Universal Robots PolyScope program: last_test_1.8.urp

ProgramRoot setBeforeStartSequence=true; directory=/programs/KINGSTON; kinematics=(a=[0, -0.425, -0.39225, 0, 0, 0], d=[0.08916, 0, 0, 0.10915, 0.09465, 0.0823], alpha=[1.5708, 0, 0, 1.5708, -1.5708, 0], deltaTheta=[0, 0, 0, 0, 0, 0], status=notInitialized); name=last_test; programVersion=(project__name=PolyScope, major__version=1, minor__version=8, svn__revision=11657, build__date=Oct 09 2013, 20:14:19); robotEnvironmentFileName=default; serialNumberRobot=2013210504
  BeforeStart description=COMMAND_SEQUENCE_BEFORE_PROGRAM_START; name=BeforeStart
    Assignment assignmentValueSource=0; expr=0; operatorValueType=INTEGER; valueSource=EXPRESSION; variable=(name=var_1, prefersPersistentValue=false, requestANewUniqueName=false)
    Assignment assignmentValueSource=0; expr=1; operatorValueType=INTEGER; valueSource=EXPRESSION; variable=(name=var_safety, prefersPersistentValue=false, requestANewUniqueName=false)
    Assignment assignmentValueSource=0; expr=50; operatorValueType=INTEGER; valueSource=EXPRESSION; variable=(name=var_force, prefersPersistentValue=false, requestANewUniqueName=false)
    Assignment assignmentValueSource=0; expr=[1,0]; operatorValueType=INTEGER; valueSource=EXPRESSION; variable=(name=var_moveType, prefersPersistentValue=false, requestANewUniqueName=false)
    Assignment assignmentValueSource=0; expr=[6,0,0,0,0,0,0]; operatorValueType=INTEGER; valueSource=EXPRESSION; variable=(name=receive_data, prefersPersistentValue=false, requestANewUniqueName=false)
    Assignment assignmentValueSource=0; expr=p[0,0,0,0,0,0]; operatorValueType=INTEGER; valueSource=EXPRESSION; variable=(name=Move_To_Pos, prefersPersistentValue=false, requestANewUniqueName=false)
    CallSubProgram subProgramNodeToCall=pose_1=get_forward_kin()
    Suppressed suppressedNode=[5,110,0,40,0,40]
    Comment 
    Suppressed suppressedNode=receive_data=socket_read_ascii_float(5)
    Assignment assignmentValueSource=0; expr=[0.2,0.2]; operatorValueType=INTEGER; valueSource=EXPRESSION; variable=(name=var_velacc, prefersPersistentValue=false, requestANewUniqueName=false)
    Script type=0; expressionBranchNode=socket_open("192.168.10.2",30000)
    Assignment assignmentValueSource=0; expr=[0,0]; operatorValueType=INTEGER; valueSource=EXPRESSION; variable=(name=task, prefersPersistentValue=false, requestANewUniqueName=false)
    Assignment assignmentValueSource=0; expr=0; operatorValueType=INTEGER; valueSource=EXPRESSION; variable=(name=coop, prefersPersistentValue=false, requestANewUniqueName=false)
  MainProgram cartesianAcceleration=1.2; cartesianSpeed=0.25; jointAcceleration=1.3962634015954636; jointSpeed=1.0471975511965976; moveAsFastAsPossible=true; sharedProcessMoveBlendRadius=0.025; featureReference=(installationNameReference=Base); motionType=JOINT_SPACE
    Suppressed suppressedNode=___tran51ate_this_name___Joint_0_name
    Suppressed suppressedNode=1
    Suppressed 
    Suppressed suppressedNode=0
    Script type=0; expressionBranchNode=ExpressionVariableNode=socket_read_ascii_float(1)
    If expr=ExpressionVariableNode[1]≟2; type=IF_NODE
      CallSubProgram subProgramNodeToCall=pose_1=get_forward_kin()
      Assignment assignmentValueSource=0; expr=[0,0]; operatorValueType=INTEGER; valueSource=EXPRESSION; variable=(name=task, prefersPersistentValue=false, requestANewUniqueName=false)
    If expr=task[1]≟3; type=ELSEIF_NODE
      Assignment assignmentValueSource=0; expr=1; operatorValueType=INTEGER; valueSource=EXPRESSION; variable=(name=coop, prefersPersistentValue=false, requestANewUniqueName=false)
      Script type=0; expressionBranchNode=socket_send_string("1")
      Assignment assignmentValueSource=0; expr=[0,0]; operatorValueType=INTEGER; valueSource=EXPRESSION; variable=(name=task, prefersPersistentValue=false, requestANewUniqueName=false)
    If expr=task[1]≟4; type=ELSEIF_NODE
      Assignment assignmentValueSource=0; expr=0; operatorValueType=INTEGER; valueSource=EXPRESSION; variable=(name=coop, prefersPersistentValue=false, requestANewUniqueName=false)
      Script type=0; expressionBranchNode=socket_send_string("1")
      Assignment assignmentValueSource=0; expr=[0,0]; operatorValueType=INTEGER; valueSource=EXPRESSION; variable=(name=task, prefersPersistentValue=false, requestANewUniqueName=false)
    If expr=task[1]≟5; type=ELSEIF_NODE
      CallSubProgram subProgramNodeToCall=receive_data=socket_read_ascii_float(2)
    If expr=task[1]≟6; type=ELSEIF_NODE
      CallSubProgram subProgramNodeToCall=receive_data=socket_read_ascii_float(2)
    If expr=task[1]≟7; type=ELSEIF_NODE
      CallSubProgram subProgramNodeToCall=receive_data=socket_read_ascii_float(2)
    If expr=task[1]≟8; type=ELSEIF_NODE
      CallSubProgram subProgramNodeToCall=receive_data=socket_read_ascii_float(5)
    If expr=task[1]≟1; type=ELSEIF_NODE
      CallSubProgram subProgramNodeToCall=receive_data=socket_read_ascii_float(6)
    Wait analogComparison=0; analogInputRange=0; analogValue=0.0; digitalValue=0; selectedAnalogSensor=-1; selectedDigitalSensor=-1; waitTime=0.01; type=TIMER_WAIT
  SubProgram name=Safety_Program
    Assignment assignmentValueSource=0; expr=0; operatorValueType=INTEGER; valueSource=EXPRESSION; variable=(name=var_safety, prefersPersistentValue=false, requestANewUniqueName=false)
    Move cartesianAcceleration=1.2; cartesianSpeed=0.25; jointAcceleration=1.3962634015954636; jointSpeed=1.0471975511965976; moveAsFastAsPossible=true; sharedProcessMoveBlendRadius=0.025; featureReference=(installationNameReference=Base); motionType=JOINT_SPACE
      Waypoint blendRadius=0.05; cartesianAcceleration=1.2; cartesianSpeed=0.25; jointAcceleration=1.3962634015954636; jointSpeed=0.10471975511965977; nextMotionTime=2.0; stoppoint=true; useSharedBlendParameter=true; position=TCP in base x=-199.996 y=-200 z=249.995 mm, rx=3.1416 ry=0 rz=0 rad; joints [-112.3, -59.43, -107.723, -102.846, 90, -202.3] deg; positionType=RELATIVE_POSITION; waypointPoseInFeatureCoordinates=(pos=(x=-0.19999561252286474, y=-0.2000002740460248, z=0.24999526084687385), rot=(x=3.1415926535838667, y=-2.8424371718740507E-6, z=-5.400202873880619E-6)); name=Waypoint_1; relativeFromJointPositionVector=(joint=[-1.96001, -1.01639, -2.01843, -1.67755, 1.5708, -3.53081], isUndefined=false); relativeFromToolAxisAngle=(x=-3.141579017620853, y=5.64237603120038E-5, z=-8.76472952232187E-6); relativeFromToolPosition=(x=-0.20000006548800986, y=-0.19998241022118884, z=0.19999450290156112)
    Halt 
  Thread name=Thread_1
    If expr=coop≟1; type=IF_NODE
      While count=0; expr=coop≟1; type=LOOP_EXPR; variable=(name=Loop_3, prefersPersistentValue=false, requestANewUniqueName=false)
        Force feature__reference=(installationNameReference=Base); force__mode__wrench=[0, 0, 0, 0, 0, 0]; limits__force=[0.15, 0.15, 0.15, 1.0472, 1.0472, 1.0472]; limits__motion=[0.1, 0.1, 0.1, 0.17453, 0.17453, 0.17453]; selection__vector=[1, 1, 1, 1, 1, 1]; type=FORCE_TYPE_FRAME
          Wait analogComparison=0; analogInputRange=0; analogValue=0.0; digitalValue=0; selectedAnalogSensor=-1; selectedDigitalSensor=-1; waitTime=0.01; type=TIMER_WAIT
      Assignment assignmentValueSource=0; expr=0; operatorValueType=INTEGER; valueSource=EXPRESSION; variable=(name=coop, prefersPersistentValue=false, requestANewUniqueName=false)
      CallSubProgram subProgramNodeToCall=pose_1=get_forward_kin()
    If type=ELSE_NODE
      If expr=ExpressionVariableNode≟1; type=IF_NODE
        If expr=ExpressionVariableNode[0]≟1; type=IF_NODE
          If checkConditionInSeperateThread=true; expr=force()<ExpressionVariableNode; type=IF_NODE
            Script type=0; expressionBranchNode=movel(Move_To_Pos,a=var_velacc[0],v=var_velacc[1],r=0)
          If type=ELSE_NODE
            CallSubProgram subProgramNodeToCall=0
        If type=ELSE_NODE
          If checkConditionInSeperateThread=true; expr=force()<ExpressionVariableNode; type=IF_NODE
            Script type=0; expressionBranchNode=movej(Move_To_Pos,a=var_velacc[0],v=var_velacc[1],r=0)
          If type=ELSE_NODE
            CallSubProgram subProgramNodeToCall=0
      Suppressed suppressedNode=movel(Move_To_Pos,a=var_velacc[0],v=var_velacc[1],r=0)
      Assignment assignmentValueSource=0; expr=ExpressionVariableNode; operatorValueType=INTEGER; valueSource=EXPRESSION; variable=(name=cur_velvac, prefersPersistentValue=false, requestANewUniqueName=false)
      Wait analogComparison=0; analogInputRange=0; analogValue=0.0; digitalValue=0; selectedAnalogSensor=-1; selectedDigitalSensor=-1; waitTime=0.01; type=TIMER_WAIT
  subProgramToCall name=SubProgram_pose
    Script type=0; expressionBranchNode=pose_1=get_forward_kin()
    Assignment assignmentValueSource=0; expr=0; operatorValueType=INTEGER; valueSource=EXPRESSION; variable=(name=pointer, prefersPersistentValue=false, requestANewUniqueName=false)
    While count=0; expr=ExpressionVariableNode<ExpressionVariableNode[0]; type=LOOP_EXPR; variable=(name=Loop_2, prefersPersistentValue=false, requestANewUniqueName=false)
      Script type=0; expressionBranchNode=Move_To_Pos[pointer]=pose_1[pointer]
      Assignment assignmentValueSource=0; expr=ExpressionVariableNode+1; operatorValueType=INTEGER; valueSource=EXPRESSION; variable=(name=pointer, prefersPersistentValue=false, requestANewUniqueName=false)
  subProgramToCall name=SubProgram_01
    Comment commentString=robot position and orientation
    Script type=0; expressionBranchNode=receive_data=socket_read_ascii_float(6)
    If expr=ExpressionVariableNode[0]≠6; type=IF_NODE
      Script type=0; expressionBranchNode=socket_send_string("0")
    If type=ELSE_NODE
      Script type=0; expressionBranchNode=socket_send_string("1")
      Assignment assignmentValueSource=0; expr=0; operatorValueType=INTEGER; valueSource=EXPRESSION; variable=(name=pointer, prefersPersistentValue=false, requestANewUniqueName=false)
      While count=0; expr=ExpressionVariableNode<ExpressionVariableNode[0]; type=LOOP_EXPR; variable=(name=Loop_4, prefersPersistentValue=false, requestANewUniqueName=false)
        Script type=0; expressionBranchNode=Move_To_Pos[pointer]=receive_data[pointer+1]
        Assignment assignmentValueSource=0; expr=ExpressionVariableNode+1; operatorValueType=INTEGER; valueSource=EXPRESSION; variable=(name=pointer, prefersPersistentValue=false, requestANewUniqueName=false)
      Assignment assignmentValueSource=0; expr=[0,0]; operatorValueType=INTEGER; valueSource=EXPRESSION; variable=(name=task, prefersPersistentValue=false, requestANewUniqueName=false)
  subProgramToCall name=SubProgram_02
    Script type=0; expressionBranchNode=pose_1=get_forward_kin()
    Script type=0; expressionBranchNode=socket_send_string(pose_1)
  subProgramToCall name=SubProgram_05
    Comment commentString=velocity and acceleration parameters
    Script type=0; expressionBranchNode=receive_data=socket_read_ascii_float(2)
    If expr=ExpressionVariableNode[0]≠2; type=IF_NODE
      Script type=0; expressionBranchNode=socket_send_string("0")
    If type=ELSE_NODE
      Script type=0; expressionBranchNode=socket_send_string("1")
      If expr=ExpressionVariableNode[1]≟ True; type=IF_NODE
        Script type=0; expressionBranchNode=digital_out[ExpressionVariableNode[2]]= True
      If type=ELSE_NODE
        Script type=0; expressionBranchNode=digital_out[ExpressionVariableNode[2]]= False
      Assignment assignmentValueSource=0; expr=[0,0]; operatorValueType=INTEGER; valueSource=EXPRESSION; variable=(name=task, prefersPersistentValue=false, requestANewUniqueName=false)
  subProgramToCall name=SubProgram_06
    Comment commentString=velocity and acceleration parameters
    Script type=0; expressionBranchNode=receive_data=socket_read_ascii_float(2)
    If expr=ExpressionVariableNode[0]≠2; type=IF_NODE
      Script type=0; expressionBranchNode=socket_send_string("0")
    If type=ELSE_NODE
      Script type=0; expressionBranchNode=socket_send_string("1")
      If expr=ExpressionVariableNode[1]≟1; type=IF_NODE
        Assignment assignmentValueSource=0; expr=[1,0]; operatorValueType=INTEGER; valueSource=EXPRESSION; variable=(name=var_moveType, prefersPersistentValue=false, requestANewUniqueName=false)
      If type=ELSE_NODE
        Assignment assignmentValueSource=0; expr=[2,0]; operatorValueType=INTEGER; valueSource=EXPRESSION; variable=(name=var_moveType, prefersPersistentValue=false, requestANewUniqueName=false)
  subProgramToCall name=SubProgram_07
    Comment commentString=velocity and acceleration parameters
    Script type=0; expressionBranchNode=receive_data=socket_read_ascii_float(2)
    If expr=ExpressionVariableNode[0]≠2; type=IF_NODE
      Script type=0; expressionBranchNode=socket_send_string("0")
    If type=ELSE_NODE
      Script type=0; expressionBranchNode=socket_send_string("1")
      Assignment assignmentValueSource=0; expr=0; operatorValueType=INTEGER; valueSource=EXPRESSION; variable=(name=pointer, prefersPersistentValue=false, requestANewUniqueName=false)
      While count=0; expr=ExpressionVariableNode<ExpressionVariableNode[0]; type=LOOP_EXPR; variable=(name=Loop_1, prefersPersistentValue=false, requestANewUniqueName=false)
        Script type=0; expressionBranchNode=var_velacc[pointer]=receive_data[pointer+1]
        Assignment assignmentValueSource=0; expr=ExpressionVariableNode+1; operatorValueType=INTEGER; valueSource=EXPRESSION; variable=(name=pointer, prefersPersistentValue=false, requestANewUniqueName=false)
      Assignment assignmentValueSource=0; expr=[0,0]; operatorValueType=INTEGER; valueSource=EXPRESSION; variable=(name=task, prefersPersistentValue=false, requestANewUniqueName=false)
  subProgramToCall name=SubProgram_08
    Comment commentString=gripper parameters
    Script type=0; expressionBranchNode=receive_data=socket_read_ascii_float(5)
    If expr=ExpressionVariableNode[0]≠5; type=IF_NODE
      Script type=0; expressionBranchNode=socket_send_string("0")
    If type=ELSE_NODE
      Script type=0; expressionBranchNode=socket_send_string("1")
      Assignment assignmentValueSource=0; expr=ExpressionVariableNode[1]; operatorValueType=INTEGER; valueSource=EXPRESSION; variable=(name=DO8_Off_DO9_Off, prefersPersistentValue=false, requestANewUniqueName=false)
      Assignment assignmentValueSource=0; expr=ExpressionVariableNode[2]; operatorValueType=INTEGER; valueSource=EXPRESSION; variable=(name=DO8_On_DO9_Off, prefersPersistentValue=false, requestANewUniqueName=false)
      Assignment assignmentValueSource=0; expr=ExpressionVariableNode[3]; operatorValueType=INTEGER; valueSource=EXPRESSION; variable=(name=DO8_Off_DO9_On, prefersPersistentValue=false, requestANewUniqueName=false)
      Assignment assignmentValueSource=0; expr=ExpressionVariableNode[4]; operatorValueType=INTEGER; valueSource=EXPRESSION; variable=(name=DO8_On_DO9_On, prefersPersistentValue=false, requestANewUniqueName=false)
      Assignment assignmentValueSource=0; expr=ExpressionVariableNode[5]; operatorValueType=INTEGER; valueSource=EXPRESSION; variable=(name=Grip_Force, prefersPersistentValue=false, requestANewUniqueName=false)
      Script type=1; cachedFileContents=if Grip_Force > 40:
        | 	Grip_Force = 40
        | 	popup("'Grip_Force' is too high - the value have been limited to  40N", title="Warning",  warning = True, error=False)
        | 	pause
        | end
        | 
        | if Grip_Force < 3:
        | 	Grip_Force = 3
        | 	popup("'Grip_Force' is too low - the value have been limited to  3N", title="Warning",  warning = True, error=False)
        | 	pause
        | end
        | 
        | if DO8_Off_DO9_Off > 110:
        | 	DO8_Off_DO9_Off = 110
        | 	popup("'DO8_Off_DO9_Off ' is too high - the value have been limited to  110mm", title="Warning",  warning = True, error=False)
        | 	pause
        | end
        | 
        | if DO8_Off_DO9_Off < 0:
        | 	DO8_Off_DO9_Off = 0
        | 	popup("'DO8_Off_DO9_Off ' is too low - the value have been limited to  0mm", title="Warning",  warning = True, error=False)
        | 	pause
        | end
        | 
        | if DO8_Off_DO9_On > 110:
        | 	DO8_Off_DO9_On = 110
        | 	popup("'DO8_Off_DO9_On ' is too high - the value have been limited to  110mm", title="Warning",  warning = True, error=False)
        | 	pause
        | end
        | 
        | if DO8_Off_DO9_On < 0:
        | 	DO8_Off_DO9_On = 0
        | 	popup("'DO8_Off_DO9_On ' is too low - the value have been limited to  0mm", title="Warning",  warning = True, error=False)
        | 	pause
        | end
        | 
        | 
        | 
        | 	
        | if DO8_On_DO9_Off > 110:
        | 	DO8_On_DO9_Off = 110
        | 	popup("'DO8_On_DO9_Off ' is too high - the value have been limited to  110mm", title="Warning",  warning = True, error=False)
        | 	pause
        | end
        | 
        | if DO8_On_DO9_Off < 0:
        | 	DO8_On_DO9_Off = 0
        | 	popup("'DO8_On_DO9_Off ' is too low - the value have been limited to  0mm", title="Warning",  warning = True, error=False)
        | 	pause
        | end
        | 
        | if DO8_On_DO9_On > 110:
        | 	DO8_On_DO9_On = 110
        | 	popup("'DO8_On_DO9_On ' is too high - the value have been limited to  110mm", title="Warning",  warning = True, error=False)
        | 	pause
        | end
        | 
        | if DO8_On_DO9_On < 0:
        | 	DO8_On_DO9_On = 0
        | 	popup("'DO8_On_DO9_On ' is too low - the value have been limited to  0mm", title="Warning",  warning = True, error=False)
        | 	pause
        | end
        | 
        | 
        | #simple mapping 
        | force0 = floor(Grip_Force)
        | pos0 = floor(DO8_On_DO9_On*10)
        | force1 = floor(Grip_Force)
        | pos1 = floor(DO8_Off_DO9_On*10)
        | force2 = floor(Grip_Force)
        | pos2 = floor(DO8_On_DO9_Off*10)
        | force3 = floor(Grip_Force)
        | pos3 = floor(DO8_Off_DO9_Off*10); scriptFile=/home/ur/ursim-3.0/programs/R1 04-01-2015/Release1.00-04-01-2015/Technical scripts/wrap1G4P1F.txt
      Script type=1; cachedFileContents=def bit_bang_spi_master_UR_script(input):
        | 	local i = 0
        | 	while i < 8:
        | 		set_digital_out(8, True)
        | 	
        | 		if input >= 128:
        | 			set_digital_out(9, False) 
        | 			input = input - 128
        | 		 else:
        | 		  	set_digital_out(9, True) 
        | 		  end  
        | 		  input = input * 2
        | 		  sleep(0.008)
        | 		  set_digital_out(8, False)
        | 		  sleep(0.008) 
        | 		  i = i + 1
        |   	end
        | end
        | 
        | 
        | 
        | version_number = 0 
        | length = 15				 
        | 
        | set_digital_out(9, False) 
        | set_digital_out(8, False)
        | set_tool_voltage(0)
        | sleep(1.5)
        | set_tool_voltage(24)
        | sleep(0.032)
        | set_tool_voltage(0)
        | sleep(0.064)
        | 
        | set_tool_voltage(24)
        | sleep(0.032)
        | set_tool_voltage(0)
        | sleep(0.064)
        | 
        | set_tool_voltage(24)
        | sleep(0.032)
        | set_tool_voltage(0)
        | sleep(0.064)
        | 
        | set_tool_voltage(24)
        | sleep(0.032)
        | set_tool_voltage(0)
        | sleep(0.064)
        | 
        | set_tool_voltage(24)
        | 
        | 
        | timeout = 0
        | while get_digital_in(8) == False:
        | 	timeout = timeout+1
        | 	sleep(0.008)
        | 	if timeout > 250:
        | 		popup("Gripper is not responding", title="Error",  warning = False, error=True)
        | 		return 1
        | 	end
        | end
        | 
        | 
        | 
        | timeout = 0
        | while get_digital_in(9):
        | 	timeout = timeout+1
        | 	sleep(0.008)
        | 	if timeout > 250:
        | 		popup("Gripper is not responding", title="Error",  warning = False, error=True)
        | 		return 1
        | 	end
        | end
        | 
        | 
        | bit_bang_spi_master_UR_script(version_number)
        | bit_bang_spi_master_UR_script(length)
        | 
        | bit_bang_spi_master_UR_script(force0)
        | bit_bang_spi_master_UR_script(pos0 - (floor(pos0/256)*256))
        | bit_bang_spi_master_UR_script(floor(pos0/256))
        | 
        | bit_bang_spi_master_UR_script(force1)
        | bit_bang_spi_master_UR_script(pos1 - (floor(pos1/256)*256))
        | bit_bang_spi_master_UR_script(floor(pos1/256))
        | 
        | bit_bang_spi_master_UR_script(force2)
        | bit_bang_spi_master_UR_script(pos2 - (floor(pos2/256)*256))
        | bit_bang_spi_master_UR_script(floor(pos2/256))
        | 
        | bit_bang_spi_master_UR_script(force3)
        | bit_bang_spi_master_UR_script(pos3 - (floor(pos3/256)*256))
        | bit_bang_spi_master_UR_script(floor(pos3/256))
        | 
        | bit_bang_spi_master_UR_script(85)
        | 
        | 
        | 
        | set_digital_out(9, False) 
        | set_digital_out(8, False)
        | 
        | timeout = 0
        | while get_digital_in(9) == True:
        | 	timeout = timeout+1
        | 	sleep(0.008)
        | 	if timeout > 250:
        | 		popup("Gripper is not responding", title="Error",  warning = False, error=True)
        | 		return 1
        | 	end
        | end
        | 
        | timeout = 0
        | while get_digital_in(9) == False:
        | 	timeout = timeout+1
        | 	sleep(0.008)
        | 	if timeout > 250:
        | 		popup("Gripper is not responding", title="Error",  warning = False, error=True)
        | 		return 1
        | 	end
        | end
        | 
        | return 0; scriptFile=/home/ur/ursim-3.0/programs/R1 04-01-2015/Script update 1.01/Technical scripts/program_gripper.txt
      Assignment assignmentValueSource=0; expr=[0,0]; operatorValueType=INTEGER; valueSource=EXPRESSION; variable=(name=task, prefersPersistentValue=false, requestANewUniqueName=false)
